// TIA Portal V20 export
FUNCTION_BLOCK "timer ON"   // FB6, LAD
{ S7_Optimized_Access := 'TRUE' }
// stored: SetENOAutomatically false
   VAR_OUTPUT
      second : Int;
      minutes : Int;
      hours : Real;
      days : Real;
      years : Real;
   END_VAR
   VAR
      P_TRIG : Bool;
      Timer_R : Bool;
   END_VAR
   VAR_TEMP
      tVKE1 : Bool;
      tVKE0 : Bool;
   END_VAR
   VAR_TEMP   // added for the SCL form of the ladder/FBD networks
      _w1 : Bool;
   END_VAR
BEGIN

REGION Network 1: Create tVKE1 Netzwek
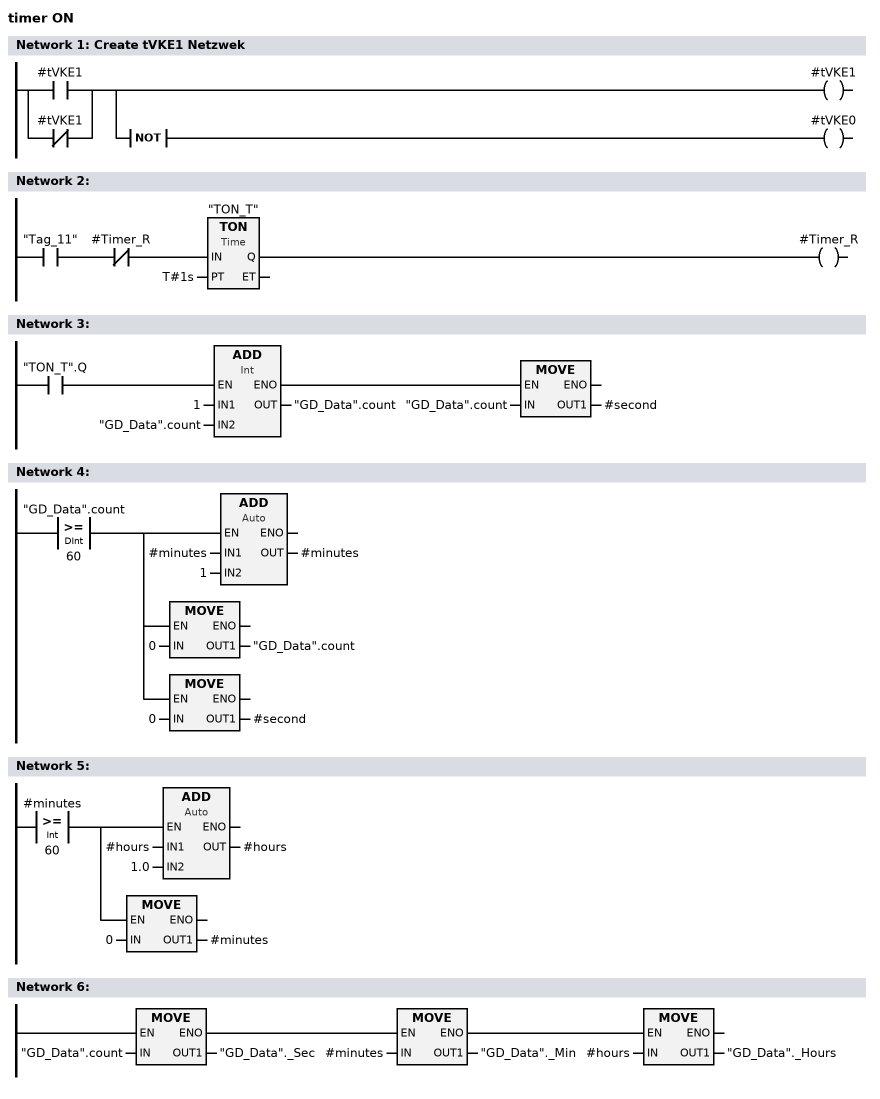
   RUNG wire#powerrail
      Contact( #tVKE1 )
      wire#w1
      Coil( #tVKE1 )
   END_RUNG
   RUNG wire#powerrail
      I_Contact( #tVKE1 )
   END_RUNG wire#w1
   RUNG wire#w1
      Not()
      Coil( #tVKE0 )
   END_RUNG
   // the same network as SCL:
   #tVKE1 := #tVKE1 OR NOT #tVKE1;
   #tVKE0 := NOT #tVKE1;
END_REGION

REGION Network 2
   RUNG wire#powerrail
      Contact( "Tag_11" )
      I_Contact( #Timer_R )
      { S7_Templates := "time_type := Time" } "TON_T".TON(pt := T#1s, et =>)
      Coil( #Timer_R )
   END_RUNG
   // the same network as SCL:
   "TON_T".TON(PT := T#1s, IN := "Tag_11" AND NOT #Timer_R);
   #Timer_R := "TON_T".Q;
END_REGION

REGION Network 3
   RUNG wire#powerrail
      Contact( "TON_T".Q )
      { S7_Templates := "SrcType := Int"; S7_GenerateENO := "TRUE" } Add(in1 := 1, in2 := "GD_Data".count, out => "GD_Data".count)
      { S7_GenerateENO := "TRUE" } Move(in := "GD_Data".count, out1 => #second)
   END_RUNG
   // the same network as SCL:
   // ENO of a box is taken as its EN; it also drops when the box reports an error
   IF "TON_T".Q THEN
       "GD_Data".count := 1 + "GD_Data".count;
       #second := "GD_Data".count;
   END_IF;
END_REGION

REGION Network 4
   RUNG wire#powerrail
      { S7_Templates := "SrcType := DInt" } GE_Contact(in1 := "GD_Data".count, in2 := 60)
      wire#w1
      { S7_GenerateENO := "TRUE" } Add(in1 := #minutes, in2 := 1, out => #minutes)
   END_RUNG
   RUNG wire#w1
      { S7_GenerateENO := "TRUE" } Move(in := 0, out1 => "GD_Data".count)
   END_RUNG
   RUNG wire#w1
      { S7_GenerateENO := "TRUE" } Move(in := 0, out1 => #second)
   END_RUNG
   // the same network as SCL:
   IF "GD_Data".count >= 60 THEN #minutes := #minutes + 1; END_IF;
   #_w1 := "GD_Data".count >= 60;
   IF #_w1 THEN
       "GD_Data".count := 0;
       #second := 0;
   END_IF;
END_REGION

REGION Network 5
   RUNG wire#powerrail
      { S7_Templates := "SrcType := Int" } GE_Contact(in1 := #minutes, in2 := 60)
      wire#w1
      { S7_GenerateENO := "TRUE" } Add(in1 := #hours, in2 := 1.0, out => #hours)
   END_RUNG
   RUNG wire#w1
      { S7_GenerateENO := "TRUE" } Move(in := 0, out1 => #minutes)
   END_RUNG
   // the same network as SCL:
   IF #minutes >= 60 THEN
       #hours := #hours + 1.0;
       #minutes := 0;
   END_IF;
END_REGION

REGION Network 6
   RUNG wire#powerrail
      { S7_GenerateENO := "TRUE" } Move(in := "GD_Data".count, out1 => "GD_Data"._Sec)
      { S7_GenerateENO := "TRUE" } Move(in := #minutes, out1 => "GD_Data"._Min)
      { S7_GenerateENO := "TRUE" } Move(in := #hours, out1 => "GD_Data"._Hours)
   END_RUNG
   // the same network as SCL:
   // ENO of a box is taken as its EN; it also drops when the box reports an error
   "GD_Data"._Sec := "GD_Data".count;
   "GD_Data"._Min := #minutes;
   "GD_Data"._Hours := #hours;
END_REGION
END_FUNCTION_BLOCK
